FUNCTION_BLOCK BuildStringInlineTest EXTENDS TcUnit.FB_TestSuite
VAR
END_VAR

BuildStringInSingleLine();

METHOD BuildStringInSingleLine : BOOL
VAR
END_VAR
TcUnit.TEST('Build string in single line');

AssertEquals_STRING(
	Expected := '12',
	Actual := BuildStringInline('1').Append('2').GetString(),
	Message := 'Should return built string');

AssertEquals_STRING(
	Expected := 'ab',
	Actual := BuildStringInline('a').Append('b').GetString(),
	Message := 'Should return another built string');

TEST_FINISHED();
END_METHOD

END_FUNCTION_BLOCK

(* stored: Version 1.1.0.1, ProductVersion 3.1.4024.15
   POU BuildStringInlineTest: Id {0ee7946b-ff3f-022f-3ed1-0529365e9ab5}, SpecialFunc None
   Method BuildStringInSingleLine: Id {aa2944c8-cf89-0007-2be6-1c371ef99030} *)
